(* This sample demonstrates how to use the UA_ConnectGetStatus function block to retrieve server status. *)
PROGRAM PRG_GETSTATUS
VAR
	(* Declarations for UA_Connect *)
	fbUA_Connect			: UA_Connect;
	SessionConnectInfo		: ST_UASessionConnectInfo;
	nConnectionHdl			: DWORD;

	(* Declarations for ConnectionGetStatus *)
	fbUA_ConnectGetStatus	: UA_ConnectGetStatus;
	eUaConnectionGetStatus	: E_UAConnectionStatus;
	eUaServerState			: E_UAServerState;
	
	(* Declarations for UA_Disconnect *)
	fbUA_Disconnect		: UA_Disconnect;

	(* Other declarations *)
	iState		: INT;
	bTest		: BOOL:= TRUE;
	bDone		: BOOL;
	bBusy		: BOOL;
	bError		: BOOL;
	nErrorID	: DWORD;
END_VAR


CASE iState OF
0:	(* idle *)
	IF bTest THEN
		bTest		:= FALSE;
		bError		:= FALSE;
		nErrorID	:= 0;

		SessionConnectInfo.tConnectTimeout 		:= T#1M;
		SessionConnectInfo.tSessionTimeout 		:= T#1M;
		SessionConnectInfo.sApplicationName		:= '';
		SessionConnectInfo.eTransportProfileUri := eUATransportProfileUri_UATcp;
		
		(* Please note: in order to successfully connect to the server, you need to trust the  
		server certificate. You can do this by moving the server certificate from the "PKI\CA\rejected" to the 
		"PKI\CA\certs\trusted" folder after the first connection attempt. *)
		SessionConnectInfo.eSecurityMode 		:= eUASecurityMsgMode_Sign_Encrypt;
		SessionConnectInfo.eSecurityPolicyUri 	:= eUASecurityPolicy_Basic256Sha256;
		
		(* If the server requires user authentication, you need to specify the user credentials as follows. *) 
		//SessionConnectInfo.stUserIdentTokenType.eUserIdentTokenType := eUAUITT_Username;
		//SessionConnectInfo.stUserIdentTokenType.sTokenParam1 := 'Administrator';
		//SessionConnectInfo.stUserIdentTokenType.sTokenParam2 := 'SomeSecurePassword';
		
		iState	:= iState + 1;
	END_IF

1:	(* Open UA session *)
	fbUA_Connect(
		Execute				:= TRUE,
		ServerURL			:= sOpcUaServerUrl,
		SessionConnectInfo	:= SessionConnectInfo,
		Timeout				:= T#2M,
		ConnectionHdl		=> nConnectionHdl
	);

	IF NOT fbUA_Connect.Busy THEN
		fbUA_Connect(Execute := FALSE);

		IF NOT fbUA_Connect.Error THEN
			(* session open *)
			iState := iState + 1;
		ELSE
			bError			:= TRUE;
			nErrorID		:= fbUA_Connect.ErrorID;
			nConnectionHdl	:= 0;
			iState 			:= 0; (* idle *)
		END_IF
	END_IF

2:	(* Query server connection status *)
	fbUA_ConnectGetStatus(
		Execute				:= TRUE,
		ConnectionHdl		:= nConnectionHdl,
		Timeout				:= T#2M,
		GetServiceLevel		:= FALSE,
		ConnectionStatus	=> eUaConnectionGetStatus,
		ServerState			=> eUaServerState
	);

	IF NOT fbUA_ConnectGetStatus.Busy THEN
		fbUA_ConnectGetStatus(Execute := FALSE);

		IF NOT fbUA_ConnectGetStatus.Error THEN
			(* session open *)
			iState := iState + 1;
		ELSE
			bError			:= TRUE;
			nErrorID		:= fbUA_Connect.ErrorID;
			nConnectionHdl	:= 0;
			iState 			:= 0; (* idle *)
		END_IF
	END_IF
	
3:	(* close session *)
	fbUA_Disconnect(
		Execute			:= TRUE,
		ConnectionHdl	:= nConnectionHdl
	);

	IF NOT fbUA_Disconnect.Busy THEN
		fbUA_Disconnect(Execute := FALSE);
		bBusy := FALSE;
		IF NOT fbUA_Disconnect.Error THEN
			(* session closed *)
			iState 		:= 0;
			IF NOT bError THEN 
				bDone 	:= TRUE;
			END_IF
		ELSE
			bError			:= TRUE;
			nErrorID		:= fbUA_Disconnect.ErrorID;
			iState 			:= 0; (* idle *)
			nConnectionHdl	:= 0;
		END_IF
	END_IF
END_CASE

END_PROGRAM

(* stored: Version 1.1.0.1
   POU PRG_GETSTATUS: Id {3c230600-8f51-44eb-8de1-1b223ccc36df}, SpecialFunc None *)
